// LS Electric XG5000 project: LAB PROJECT_190021302,304,308,312
// PLC NewPLC

PROGRAM NewProgram (task: Scan Program)

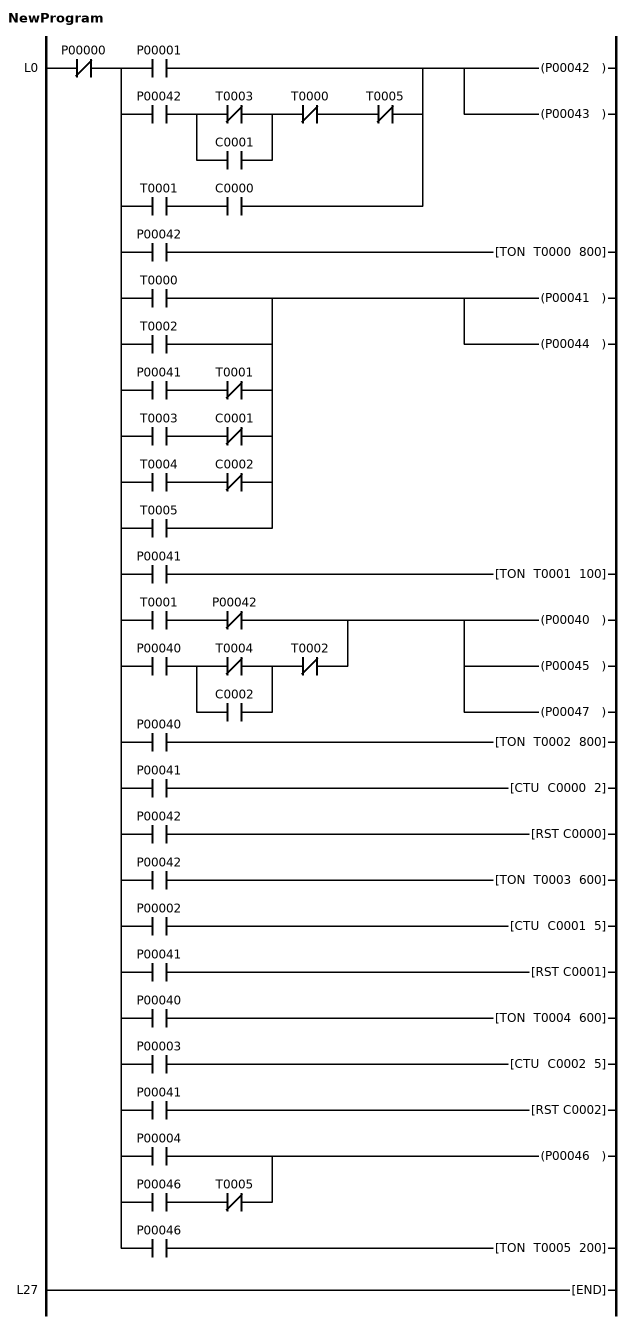
; L0
LOAD NOT  P00000
MPUSH
LOAD      P00001
LOAD      P00042
LOAD NOT  T0003
OR        C0001
AND LOAD
AND NOT   T0000
AND NOT   T0005
OR LOAD
LOAD      T0001
AND       C0000
OR LOAD
AND LOAD
OUT       P00042
OUT       P00043
MLOAD
AND       P00042
TON       T0000 800
MLOAD
LOAD      T0000
OR        T0002
LOAD      P00041
AND NOT   T0001
OR LOAD
LOAD      T0003
AND NOT   C0001
OR LOAD
LOAD      T0004
AND NOT   C0002
OR LOAD
OR        T0005
AND LOAD
OUT       P00041
OUT       P00044
MLOAD
AND       P00041
TON       T0001 100
MLOAD
LOAD      T0001
AND NOT   P00042
LOAD      P00040
LOAD NOT  T0004
OR        C0002
AND LOAD
AND NOT   T0002
OR LOAD
AND LOAD
OUT       P00040
OUT       P00045
OUT       P00047
MLOAD
AND       P00040
TON       T0002 800
MLOAD
AND       P00041
CTU       C0000 2
MLOAD
AND       P00042
RST       C0000
MLOAD
AND       P00042
TON       T0003 600
MLOAD
AND       P00002
CTU       C0001 5
MLOAD
AND       P00041
RST       C0001
MLOAD
AND       P00040
TON       T0004 600
MLOAD
AND       P00003
CTU       C0002 5
MLOAD
AND       P00041
RST       C0002
MLOAD
LOAD      P00004
LOAD      P00046
AND NOT   T0005
OR LOAD
AND LOAD
OUT       P00046
MPOP
AND       P00046
TON       T0005 200
// output comment: 
// output comment: 
; L27
END